TYPE enum_E :
(
	elit_gopickup,
	elit_init0,
	elit_init1,
	elit_init2,
	elit_init3,
	elit_init4,
	elit_init5,
	elit_init6,
	elit_init7,
	elit_init8,
	elit_init9,
	elit_init_error,
	elit_init_ok,
	elit_init_sensor_check,
	elit_initialized,
	elit_running,
	elit_starting,
	elit_wait_init,
	elit_wait_start
);
END_TYPE

(* stored: Version 1.1.0.1, ProductVersion 3.1.4022.18
   DUT enum_E: Id {21c2615d-566b-4781-ac49-c8382d9e50cd} *)
